// TIA Portal V20 export
VAR_GLOBAL   // PLC tag table "ConvConstant"
END_VAR
VAR_GLOBAL CONSTANT   // user constants
   gMinA1 : Int := 1001;
   gMaxA1 : Int := 1002;
   gMinB1 : Int := 2001;
   gMaxB1 : Int := 2002;
   gMinC1 : Int := 3001;
   gMaxC1 : Int := 3054;
   gMinD1 : Int := 4001;
   gMaxD1 : Int := 4002;
END_VAR
